SUBAPPLICATION Uebung_004b3b_AX (* Zwei gegenseitig verriegelte Toggle-Flip-Flops (Radio-Button-Logik) via Event-Verdrahtung *)
  (* Standard: 61499-2; Description: Copyright (c) 2023 Meisterschulen am Ostbahnhof This program and the accompanying materials are made available under the terms of the Eclipse Public License 2.0 which is available at https://www.eclipse.org/legal/epl-2.0/ SPDX-License-Identifier: EPL-2.0 *)
  (* Version 1.0, 2023-10-23, Franz Höpfinger, Meisterschulen am Ostbahnhof, initial API and implementation and/or initial documentation *)
  PACKAGE Uebungen;
  IMPORT logiBUS::io::DI::logiBUS_DI::Input_I1;
  IMPORT logiBUS::io::DI::logiBUS_DI::Input_I2;
  IMPORT logiBUS::io::DI::logiBUS_DI_Events::BUTTON_SINGLE_CLICK;
  IMPORT logiBUS::io::DQ::logiBUS_DO::Output_Q1;
  IMPORT logiBUS::io::DQ::logiBUS_DO::Output_Q2;
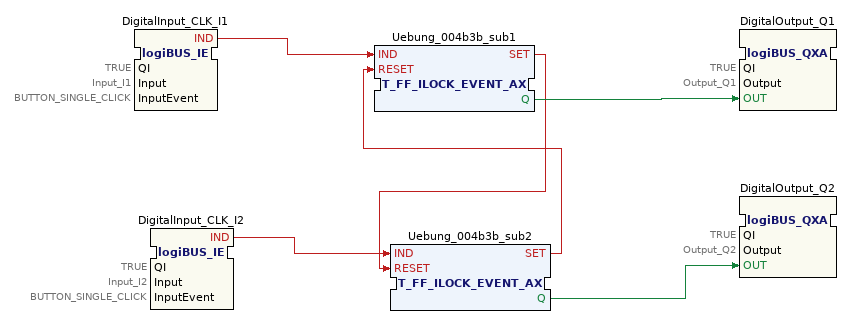
  FBS
    DigitalOutput_Q1 : logiBUS::io::DQ::logiBUS_QXA(QI := TRUE, Output := Output_Q1);
    DigitalInput_CLK_I1 : logiBUS::io::DI::logiBUS_IE(QI := TRUE, Input := Input_I1, InputEvent := BUTTON_SINGLE_CLICK);
    DigitalOutput_Q2 : logiBUS::io::DQ::logiBUS_QXA(QI := TRUE, Output := Output_Q2);
    DigitalInput_CLK_I2 : logiBUS::io::DI::logiBUS_IE(QI := TRUE, Input := Input_I2, InputEvent := BUTTON_SINGLE_CLICK);
  END_FBS
  SUBAPPS
    Uebung_004b3b_sub1 : MyLib::sys::T_FF_ILOCK_EVENT_AX;
    Uebung_004b3b_sub2 : MyLib::sys::T_FF_ILOCK_EVENT_AX;
  END_SUBAPPS
  EVENT_CONNECTIONS
    DigitalInput_CLK_I2.IND TO Uebung_004b3b_sub2.IND;
    DigitalInput_CLK_I1.IND TO Uebung_004b3b_sub1.IND;
    Uebung_004b3b_sub2.SET TO Uebung_004b3b_sub1.RESET;
    Uebung_004b3b_sub1.SET TO Uebung_004b3b_sub2.RESET;
  END_CONNECTIONS
  ADAPTER_CONNECTIONS
    Uebung_004b3b_sub1.Q TO DigitalOutput_Q1.OUT;
    Uebung_004b3b_sub2.Q TO DigitalOutput_Q2.OUT;
  END_CONNECTIONS
END_SUBAPPLICATION
